{attribute 'qualified_only'}
{attribute 'strict'}
TYPE E_Order :
(
	ASCENDING,
	DESCENDING
);
END_TYPE

(* stored: Version 1.1.0.1, ProductVersion 3.1.4024.11
   EnumerationTextList E_Order: Id {3cf6c5eb-3131-412c-80a0-0274fd4e6e1b} *)
